FUNCTION F_ConsumeTime
VAR_INPUT
	Us		:UDINT;
END_VAR
VAR
		tCurr, tEnd : T_DCTIME64;
END_VAR

tCurr := F_GetActualDcTime64();
tEnd  := tCurr + (Us * EC_DCTIME_TICKSPERMSEC64 / 1000);
WHILE (tCurr < tEnd) DO
	tCurr := F_GetActualDcTime64();
END_WHILE

END_FUNCTION

(* stored: Version 1.1.0.1, ProductVersion 3.1.4026.18
   POU F_ConsumeTime: Id {49cb8b8a-c78c-47a9-ab20-41df7c957ff9}, SpecialFunc None *)
